{attribute 'enable_dynamic_creation'}
FUNCTION_BLOCK FB_CompositeCommand IMPLEMENTS I_Command
VAR
	invoker : I_CommandInvoker;
	_Description : STRING;
	
	started : BOOL;
END_VAR

{attribute 'monitoring' := 'call'}
PROPERTY Description : STRING
GET
Description := _Description;
END_GET
END_PROPERTY

METHOD Execute : E_ProgressStatus
IF (NOT started) THEN
	started := TRUE;
	
	invoker.Reset();
	invoker.Start();
END_IF

invoker.Cyclic();

Execute := invoker.ProgressState;
END_METHOD

//FB_Init is always available implicitly and it is used primarily for initialization.
//The return value is not evaluated. For a specific influence, you can also declare the
//methods explicitly and provide additional code there with the standard initialization
//code. You can evaluate the return value.
METHOD FB_Init: BOOL
VAR_INPUT
    bInitRetains: BOOL; // TRUE: the retain variables are initialized (reset warm / reset cold)
    bInCopyCode: BOOL;  // TRUE: the instance will be copied to the copy code afterward (online change)   
	
	invoker : I_CommandInvoker;
	description : STRING;
END_VAR
THIS^.invoker := invoker;
_Description := description;
END_METHOD

METHOD Reset
VAR_INPUT
END_VAR
started := FALSE;
invoker.Reset();
END_METHOD

END_FUNCTION_BLOCK

(* stored: Version 1.1.0.1
   POU FB_CompositeCommand: Id {75a465cc-b612-40c5-93a3-8e74036cc90d}, SpecialFunc None
   Property Description: Id {fb4725b7-6b63-41d2-94b7-662c458c8703}
   Get Get: Id {5d4f5ff9-70e7-47c0-99c7-e4b9a4fd067e}
   Method Execute: Id {0243d9c3-512c-45c5-b801-d0dbdb15436d}
   Method FB_Init: Id {af1294e3-7020-4014-b09a-224e3070ddee}
   Method Reset: Id {5561878b-f7fa-4f12-9b9c-9cdff62ae017} *)
